(* Logix 5000 project; controller traffic_light_sequencer vendor 1 type 14 code 196 rev 36.11; software revision 36.00 *)

TASK MainTask (continuous, watchdog 500 ms) : MainProgram, Traffic_Light_Sequencer

MODULES
   Local : vendor 1 type 14 code 196 (5069 0, rev 36.11)
END_MODULES

VAR_GLOBAL   (* controller tags *)
   Mode_Maintenance : BOOL;
   Mode_Manual : BOOL;
   Mode_Normal : BOOL;
   PB_ManualAdvance : BOOL;
   PB_Pedestrian : BOOL;
   PB_Reset : BOOL;
   SW_MaintenanceMode : BOOL;
   SW_ManualMode : BOOL := 1;
END_VAR

PROGRAM MainProgram   (* main routine MainRoutine *)

ROUTINE MainRoutine   (* ladder *)
END_ROUTINE
END_PROGRAM

PROGRAM Traffic_Light_Sequencer   (* main routine MainRoutine *)
VAR
   EW_Green : BOOL;
   EW_Red : BOOL;
   EW_Yellow : BOOL;
   Fault_ConflictingGreens : BOOL;
   Fault_EW_MultipleLampsOn : BOOL;
   Fault_General : BOOL;
   Fault_InvalidPedState : BOOL;
   Fault_NS_MultpleLampsOn : BOOL;
   FlashBit : BOOL;
   MainExitHoldActive : BOOL;
   ManualAdvanceONS_Mem : BOOL;
   ManualAdvancePulse : BOOL;
   NS_Green : BOOL;
   NS_Red : BOOL;
   NS_Yellow : BOOL;
   PED_DontWalk : BOOL;
   PED_Walk : BOOL;
   PedReqLatched : BOOL;
   PedReqONS_Mem : BOOL;
   SeqStep : DINT;
   Status_AllRedState : BOOL;
   Status_EWActive : BOOL;
   Status_FlashYellowActive : BOOL;
   Status_NSActive : BOOL;
   Status_PedRequestPending : BOOL;
   Status_SequenceRunning : BOOL;
   Step10DoneONS_Mem : BOOL;
   Step20DoneONS_Mem : BOOL;
   Step30_TransitionPulse : BOOL;
   Step30DoneONS_Mem : BOOL;
   Step35_TransitionPulse : BOOL;
   Step35DoneONS_Mem : BOOL;
   Step40DoneONS_Mem : BOOL;
   Step50DoneONS_Mem : BOOL;
   Step60_TransitionPlus : BOOL;
   Step60DoneONS_Mem : BOOL;
   Step65_TransitionPulse : BOOL;
   Step65DoneONS : BOOL;
   T_AllRed_1 : TIMER := (PRE := 1000);
        .PRE   // 1000
   T_AllRed_2 : TIMER := (PRE := 1000);
        .PRE   // 1000
   T_EW_Green : TIMER := (PRE := 8000);
        .PRE   // 8000
   T_EW_Yellow : TIMER := (PRE := 3000);
        .PRE   // 3000
   T_FlashYellow : TIMER := (PRE := 500);
        .PRE   // 500
   T_MaintExitHold : TIMER := (PRE := 1000);
        .PRE   // 1000
   T_NS_Green : TIMER := (PRE := 8000);
        .PRE   // 8000
   T_NS_Yellow : TIMER := (PRE := 8000);
        .PRE   // 3000
   T_PedWalk_1 : TIMER := (PRE := 5000);
        .PRE   // 5000
   T_PedWalk_2 : TIMER := (PRE := 5000);
        .PRE   // 5000
END_VAR

ROUTINE Diagnostic_Status   (* ladder *)
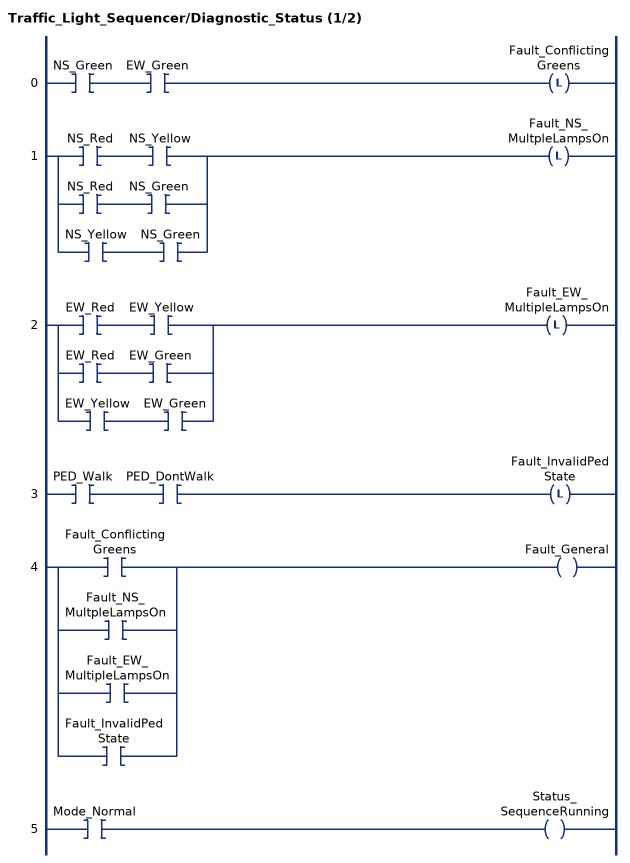
   0: XIC(NS_Green)XIC(EW_Green)OTL(Fault_ConflictingGreens);
   1: [XIC(NS_Red) XIC(NS_Yellow) ,XIC(NS_Red) XIC(NS_Green) ,XIC(NS_Yellow) XIC(NS_Green) ]OTL(Fault_NS_MultpleLampsOn);
   2: [XIC(EW_Red) XIC(EW_Yellow) ,XIC(EW_Red) XIC(EW_Green) ,XIC(EW_Yellow) XIC(EW_Green) ]OTL(Fault_EW_MultipleLampsOn);
   3: XIC(PED_Walk)XIC(PED_DontWalk)OTL(Fault_InvalidPedState);
   4: [XIC(Fault_ConflictingGreens) ,XIC(Fault_NS_MultpleLampsOn) ,XIC(Fault_EW_MultipleLampsOn) ,XIC(Fault_InvalidPedState) ]OTE(Fault_General);
   5: XIC(Mode_Normal)OTE(Status_SequenceRunning);
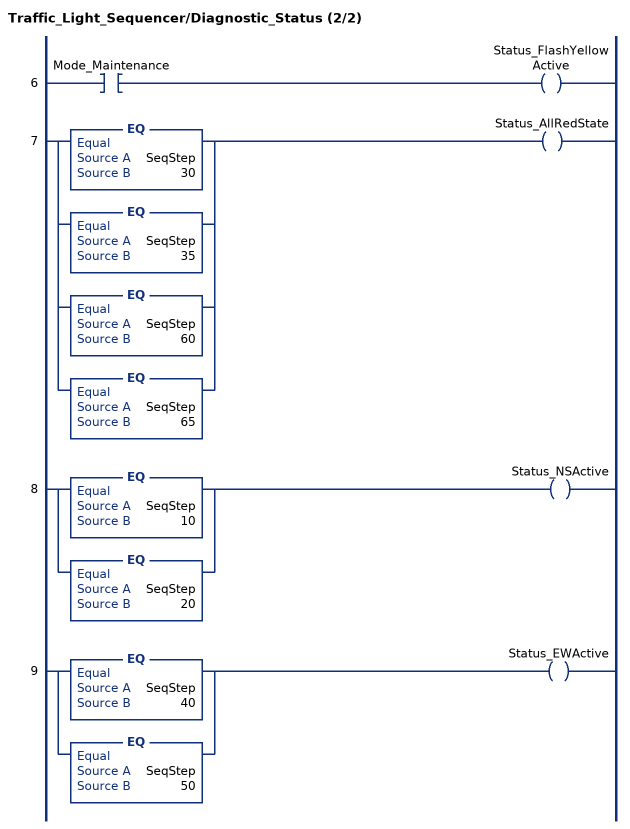
   6: XIC(Mode_Maintenance)OTE(Status_FlashYellowActive);
   7: [EQ(SeqStep,30) ,EQ(SeqStep,35) ,EQ(SeqStep,60) ,EQ(SeqStep,65) ]OTE(Status_AllRedState);
   8: [EQ(SeqStep,10) ,EQ(SeqStep,20) ]OTE(Status_NSActive);
   9: [EQ(SeqStep,40) ,EQ(SeqStep,50) ]OTE(Status_EWActive);
END_ROUTINE

ROUTINE Input_Mode_Handling   (* ladder *)
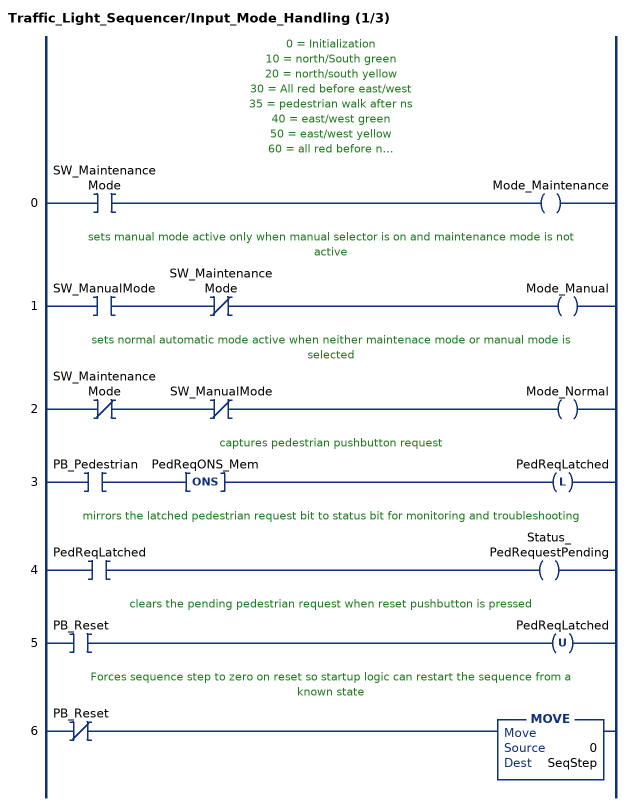
   // 0 = Initialization
   // 10 = north/South green
   // 20 = north/south yellow
   // 30 = All red before east/west
   // 35 = pedestrian walk after ns
   // 40 = east/west green
   // 50 = east/west yellow
   // 60 = all red before ns
   // 65 = Pedestrian walk after ew
   // sets maintenance mode active when the maintenance selector input is on
   0: XIC(SW_MaintenanceMode)OTE(Mode_Maintenance);
   // sets manual mode active only when manual selector is on and maintenance mode is not active
   1: XIC(SW_ManualMode)XIO(SW_MaintenanceMode)OTE(Mode_Manual);
   // sets normal automatic mode active when neither maintenace mode or manual mode is selected
   2: XIO(SW_MaintenanceMode)XIO(SW_ManualMode)OTE(Mode_Normal);
   // captures pedestrian pushbutton request
   3: XIC(PB_Pedestrian)ONS(PedReqONS_Mem)OTL(PedReqLatched);
   // mirrors the latched pedestrian request bit to status bit for monitoring and troubleshooting
   4: XIC(PedReqLatched)OTE(Status_PedRequestPending);
   // clears the pending pedestrian request when reset pushbutton is pressed
   5: XIC(PB_Reset)OTU(PedReqLatched);
   // Forces sequence step to zero on reset so startup logic can restart the sequence from a known state
   6: XIO(PB_Reset)MOVE(0,SeqStep);
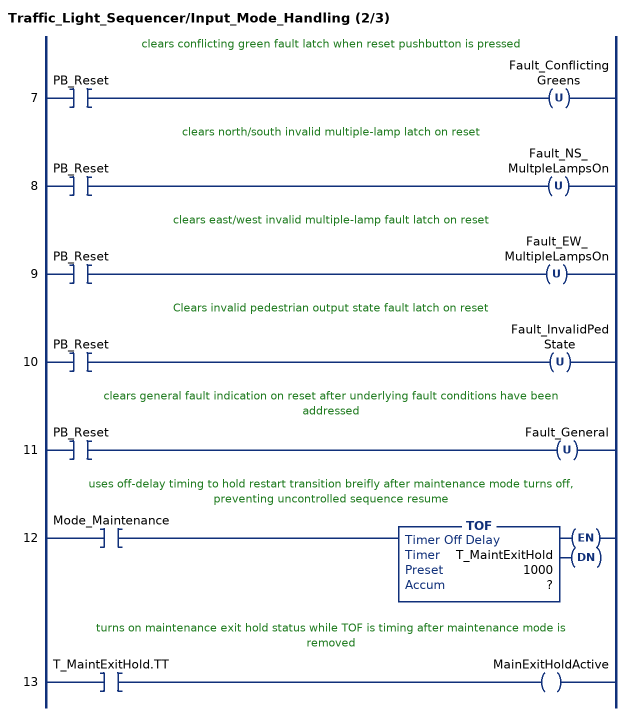
   // clears conflicting green fault latch when reset pushbutton is pressed
   7: XIC(PB_Reset)OTU(Fault_ConflictingGreens);
   // clears north/south invalid multiple-lamp latch on reset
   8: XIC(PB_Reset)OTU(Fault_NS_MultpleLampsOn);
   // clears east/west invalid multiple-lamp fault latch on reset
   9: XIC(PB_Reset)OTU(Fault_EW_MultipleLampsOn);
   // Clears invalid pedestrian output state fault latch on reset
   10: XIC(PB_Reset)OTU(Fault_InvalidPedState);
   // clears general fault indication on reset after underlying fault conditions have been addressed
   11: XIC(PB_Reset)OTU(Fault_General);
   // uses off-delay timing to hold restart transition breifly after maintenance mode turns off, preventing uncontrolled sequence resume
   12: XIC(Mode_Maintenance)TOF(T_MaintExitHold,?,?);
   // turns on maintenance exit hold status while TOF is timing after maintenance mode is removed
   13: XIC(T_MaintExitHold.TT)OTE(MainExitHoldActive);
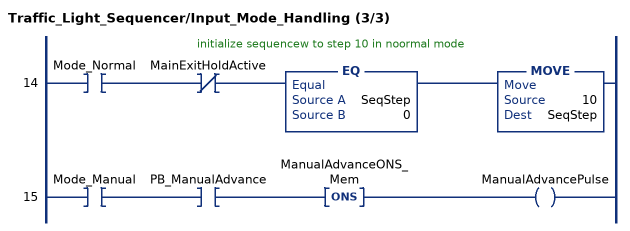
   // initialize sequencew to step 10 in noormal mode
   14: XIC(Mode_Normal)XIO(MainExitHoldActive)EQ(SeqStep,0)MOVE(10,SeqStep);
   15: XIC(Mode_Manual)XIC(PB_ManualAdvance)ONS(ManualAdvanceONS_Mem)OTE(ManualAdvancePulse);
END_ROUTINE

ROUTINE MainRoutine   (* ladder *)
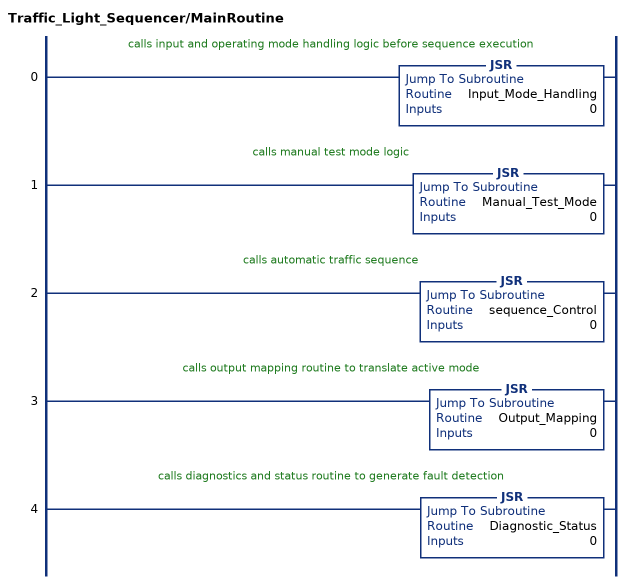
   // calls input and operating mode handling logic before sequence execution
   0: JSR(Input_Mode_Handling,0);
   // calls manual test mode logic
   1: JSR(Manual_Test_Mode,0);
   // calls automatic traffic sequence
   2: JSR(sequence_Control,0);
   // calls output mapping routine to translate active mode
   3: JSR(Output_Mapping,0);
   // calls diagnostics and status routine to generate fault detection
   4: JSR(Diagnostic_Status,0);
END_ROUTINE

ROUTINE Manual_Test_Mode   (* ladder *)
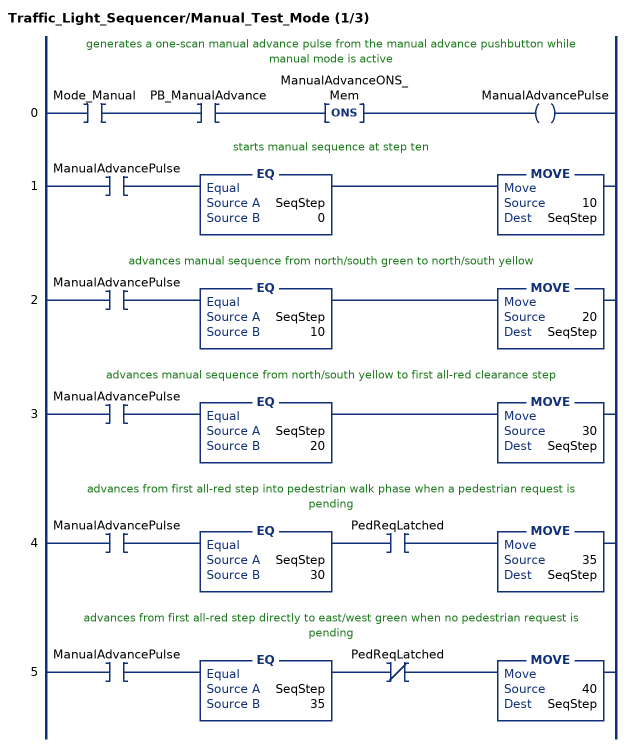
   // generates a one-scan manual advance pulse from the manual advance pushbutton while manual mode is active
   0: XIC(Mode_Manual)XIC(PB_ManualAdvance)ONS(ManualAdvanceONS_Mem)OTE(ManualAdvancePulse);
   // starts manual sequence at step ten
   1: XIC(ManualAdvancePulse)EQ(SeqStep,0)MOVE(10,SeqStep);
   // advances manual sequence from north/south green to north/south yellow
   2: XIC(ManualAdvancePulse)EQ(SeqStep,10)MOVE(20,SeqStep);
   // advances manual sequence from north/south yellow to first all-red clearance step
   3: XIC(ManualAdvancePulse)EQ(SeqStep,20)MOVE(30,SeqStep);
   // advances from first all-red step into pedestrian walk phase when a pedestrian request is pending
   4: XIC(ManualAdvancePulse)EQ(SeqStep,30)XIC(PedReqLatched)MOVE(35,SeqStep);
   // advances from first all-red step directly to east/west green when no pedestrian request is pending
   5: XIC(ManualAdvancePulse)EQ(SeqStep,35)XIO(PedReqLatched)MOVE(40,SeqStep);
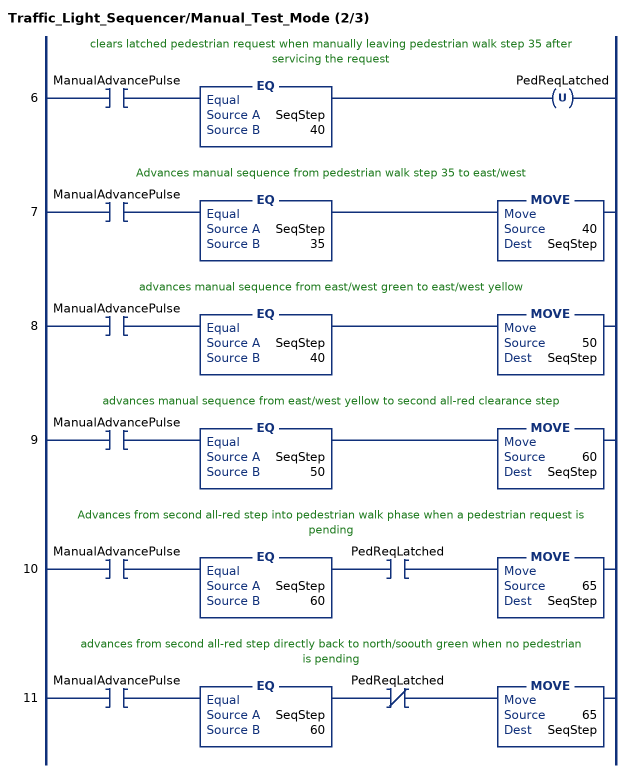
   // clears latched pedestrian request when manually leaving pedestrian walk step 35 after servicing the request
   6: XIC(ManualAdvancePulse)EQ(SeqStep,40)OTU(PedReqLatched);
   // Advances manual sequence from pedestrian walk step 35 to east/west
   7: XIC(ManualAdvancePulse)EQ(SeqStep,35)MOVE(40,SeqStep);
   // advances manual sequence from east/west green to east/west yellow
   8: XIC(ManualAdvancePulse)EQ(SeqStep,40)MOVE(50,SeqStep);
   // advances manual sequence from east/west yellow to second all-red clearance step
   9: XIC(ManualAdvancePulse)EQ(SeqStep,50)MOVE(60,SeqStep);
   // Advances from second all-red step into pedestrian walk phase when a pedestrian request is pending
   10: XIC(ManualAdvancePulse)EQ(SeqStep,60)XIC(PedReqLatched)MOVE(65,SeqStep);
   // advances from second all-red step directly back to north/soouth green when no pedestrian is pending
   11: XIC(ManualAdvancePulse)EQ(SeqStep,60)XIO(PedReqLatched)MOVE(65,SeqStep);
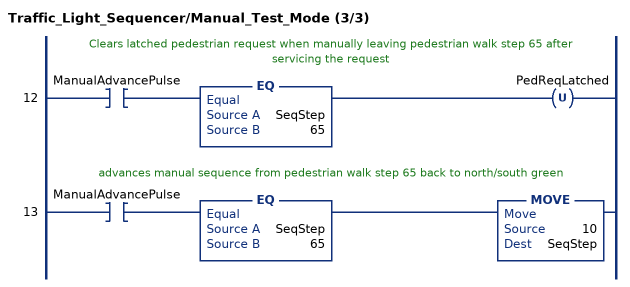
   // Clears latched pedestrian request when manually leaving pedestrian walk step 65 after servicing the request
   12: XIC(ManualAdvancePulse)EQ(SeqStep,65)OTU(PedReqLatched);
   // advances manual sequence from pedestrian walk step 65 back to north/south green
   13: XIC(ManualAdvancePulse)EQ(SeqStep,65)MOVE(10,SeqStep);
END_ROUTINE

ROUTINE Output_Mapping   (* ladder *)
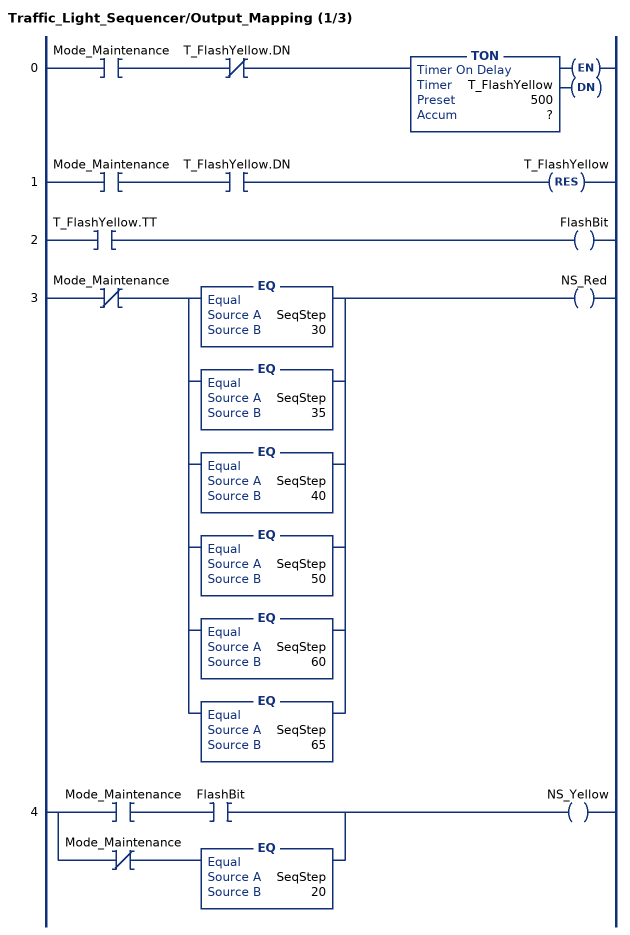
   0: XIC(Mode_Maintenance)XIO(T_FlashYellow.DN)TON(T_FlashYellow,?,?);
   1: XIC(Mode_Maintenance)XIC(T_FlashYellow.DN)RES(T_FlashYellow);
   2: XIC(T_FlashYellow.TT)OTE(FlashBit);
   3: XIO(Mode_Maintenance)[EQ(SeqStep,30) ,EQ(SeqStep,35) ,EQ(SeqStep,40) ,EQ(SeqStep,50) ,EQ(SeqStep,60) ,EQ(SeqStep,65) ]OTE(NS_Red);
   4: [XIC(Mode_Maintenance) XIC(FlashBit) ,XIO(Mode_Maintenance) EQ(SeqStep,20) ]OTE(NS_Yellow);
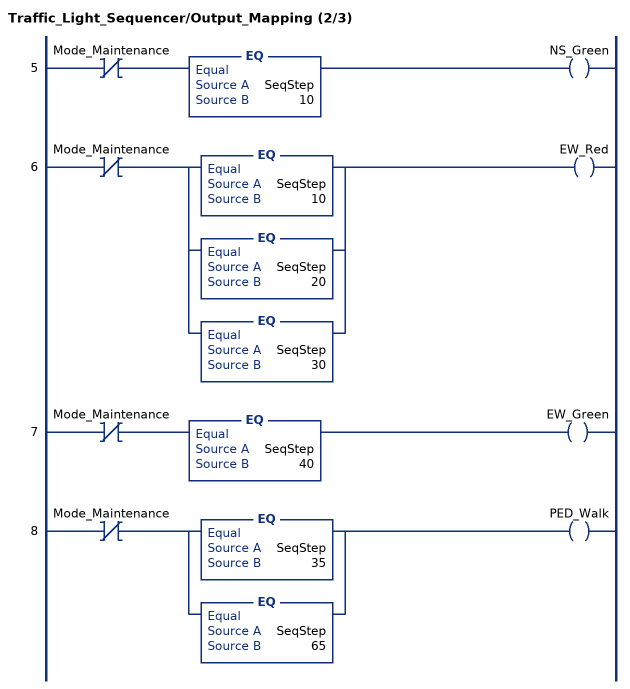
   5: XIO(Mode_Maintenance)EQ(SeqStep,10)OTE(NS_Green);
   6: XIO(Mode_Maintenance)[EQ(SeqStep,10) ,EQ(SeqStep,20) ,EQ(SeqStep,30) ]OTE(EW_Red);
   7: XIO(Mode_Maintenance)EQ(SeqStep,40)OTE(EW_Green);
   8: XIO(Mode_Maintenance)[EQ(SeqStep,35) ,EQ(SeqStep,65) ]OTE(PED_Walk);
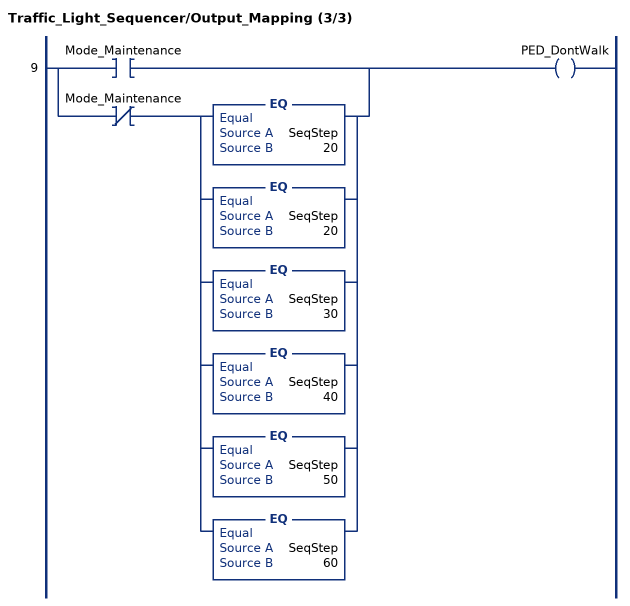
   9: [XIC(Mode_Maintenance) ,XIO(Mode_Maintenance) [EQ(SeqStep,20) ,EQ(SeqStep,20) ,EQ(SeqStep,30) ,EQ(SeqStep,40) ,EQ(SeqStep,50) ,EQ(SeqStep,60) ] ]OTE(PED_DontWalk);
END_ROUTINE

ROUTINE sequence_Control   (* ladder *)
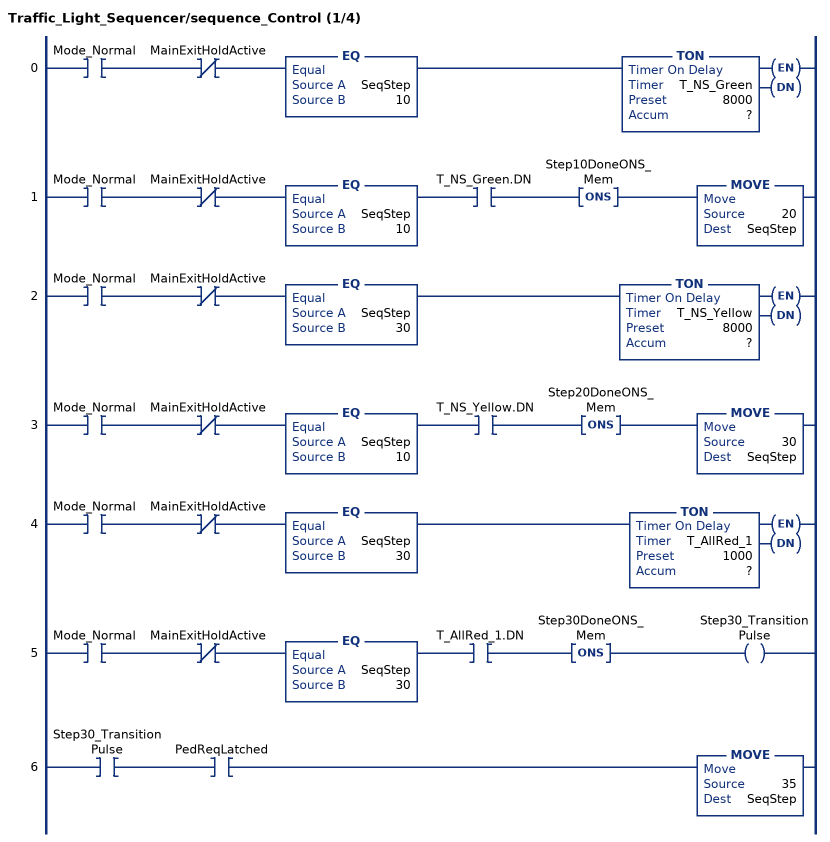
   0: XIC(Mode_Normal)XIO(MainExitHoldActive)EQ(SeqStep,10)TON(T_NS_Green,?,?);
   1: XIC(Mode_Normal)XIO(MainExitHoldActive)EQ(SeqStep,10)XIC(T_NS_Green.DN)ONS(Step10DoneONS_Mem)MOVE(20,SeqStep);
   2: XIC(Mode_Normal)XIO(MainExitHoldActive)EQ(SeqStep,30)TON(T_NS_Yellow,?,?);
   3: XIC(Mode_Normal)XIO(MainExitHoldActive)EQ(SeqStep,10)XIC(T_NS_Yellow.DN)ONS(Step20DoneONS_Mem)MOVE(30,SeqStep);
   4: XIC(Mode_Normal)XIO(MainExitHoldActive)EQ(SeqStep,30)TON(T_AllRed_1,?,?);
   5: XIC(Mode_Normal)XIO(MainExitHoldActive)EQ(SeqStep,30)XIC(T_AllRed_1.DN)ONS(Step30DoneONS_Mem)OTE(Step30_TransitionPulse);
   6: XIC(Step30_TransitionPulse)XIC(PedReqLatched)MOVE(35,SeqStep);
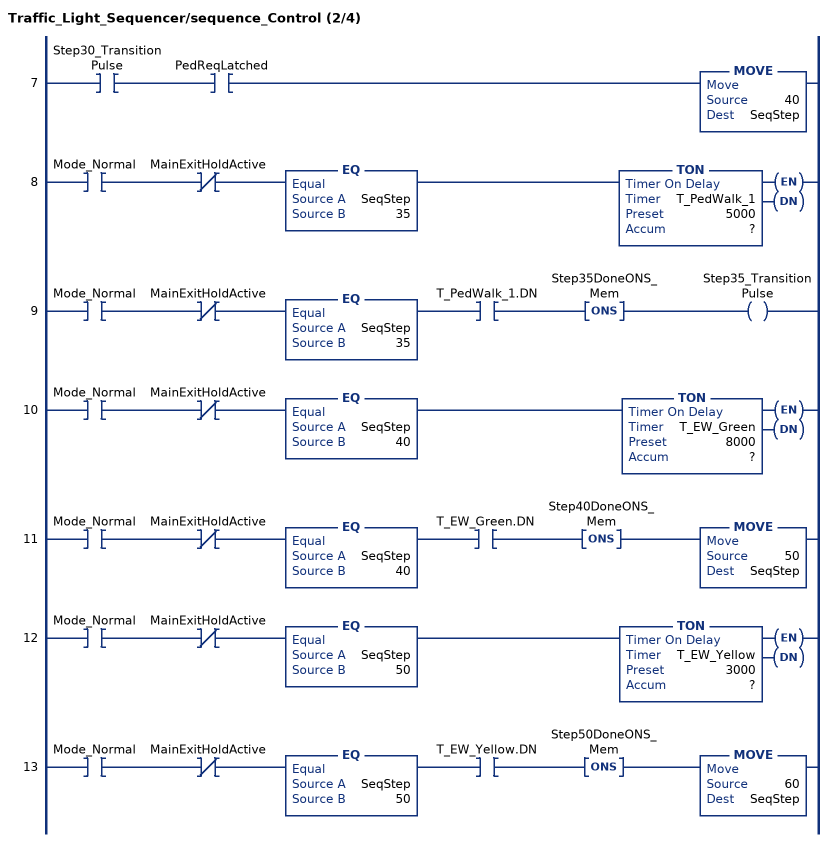
   7: XIC(Step30_TransitionPulse)XIC(PedReqLatched)MOVE(40,SeqStep);
   8: XIC(Mode_Normal)XIO(MainExitHoldActive)EQ(SeqStep,35)TON(T_PedWalk_1,?,?);
   9: XIC(Mode_Normal)XIO(MainExitHoldActive)EQ(SeqStep,35)XIC(T_PedWalk_1.DN)ONS(Step35DoneONS_Mem)OTE(Step35_TransitionPulse);
   10: XIC(Mode_Normal)XIO(MainExitHoldActive)EQ(SeqStep,40)TON(T_EW_Green,?,?);
   11: XIC(Mode_Normal)XIO(MainExitHoldActive)EQ(SeqStep,40)XIC(T_EW_Green.DN)ONS(Step40DoneONS_Mem)MOVE(50,SeqStep);
   12: XIC(Mode_Normal)XIO(MainExitHoldActive)EQ(SeqStep,50)TON(T_EW_Yellow,?,?);
   13: XIC(Mode_Normal)XIO(MainExitHoldActive)EQ(SeqStep,50)XIC(T_EW_Yellow.DN)ONS(Step50DoneONS_Mem)MOVE(60,SeqStep);
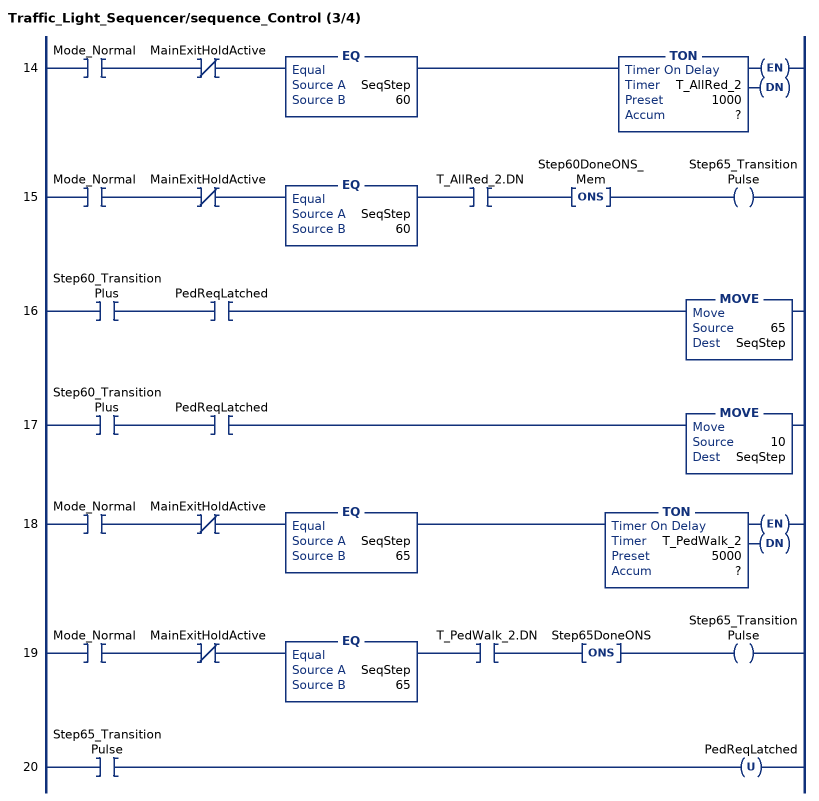
   14: XIC(Mode_Normal)XIO(MainExitHoldActive)EQ(SeqStep,60)TON(T_AllRed_2,?,?);
   15: XIC(Mode_Normal)XIO(MainExitHoldActive)EQ(SeqStep,60)XIC(T_AllRed_2.DN)ONS(Step60DoneONS_Mem)OTE(Step65_TransitionPulse);
   16: XIC(Step60_TransitionPlus)XIC(PedReqLatched)MOVE(65,SeqStep);
   17: XIC(Step60_TransitionPlus)XIC(PedReqLatched)MOVE(10,SeqStep);
   18: XIC(Mode_Normal)XIO(MainExitHoldActive)EQ(SeqStep,65)TON(T_PedWalk_2,?,?);
   19: XIC(Mode_Normal)XIO(MainExitHoldActive)EQ(SeqStep,65)XIC(T_PedWalk_2.DN)ONS(Step65DoneONS)OTE(Step65_TransitionPulse);
   20: XIC(Step65_TransitionPulse)OTU(PedReqLatched);
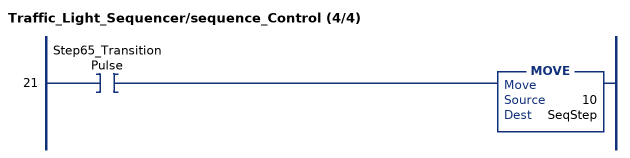
   21: XIC(Step65_TransitionPulse)MOVE(10,SeqStep);
END_ROUTINE
END_PROGRAM
